// TIA Portal project "trafik_lamba_uygulama_sim" (V14)

(* hardware
DEVICE "S71500/ET200MP station_1"  S7-1500 station
   slot 0: "Rail_0"  Rack  6ES7 590-1***0-0AA0
   slot 1: "PLC_1"  CPU 1511C-1 PN  6ES7 511-1CK00-0AB0  V2.0
      slot 3: "CPU display_1"  6ES7591-1AA00-0AA0
*)

// ===== PLC "PLC_1"  CPU 1511C-1 PN =====

VAR_GLOBAL   // PLC tag table "Default tag table"
   ""start"" AT %I0.1 : Bool;
   ""reset"" AT %I0.0 : Bool;
   ""yol_1-3"" AT %Q0.0 : Bool;
   ""yol_2-4"" AT %Q0.1 : Bool;
   ""kirmizi_isik_yol-1"" AT %Q1.0 : Bool;
   ""sari_isik_yol-1"" AT %Q1.1 : Bool;
   ""yesil_isik_yol-1"" AT %Q1.2 : Bool;
   ""kirmizi_isik_yol-3"" AT %Q1.3 : Bool;
   ""sari_isik_yol-3"" AT %Q1.4 : Bool;
   ""yesil_isik_yol-3"" AT %Q1.5 : Bool;
   ""yol_5-6"" AT %Q0.2 : Bool;
   ""kirmizi_isik_yol-2"" AT %Q2.0 : Bool;
   ""sari_isik_yol-2"" AT %Q2.1 : Bool;
   ""yesil_isik_yol-2"" AT %Q2.2 : Bool;
   ""kirmizi_isik_yol-4"" AT %Q2.3 : Bool;
   ""sari_isik_yol-4"" AT %Q2.4 : Bool;
   ""yesil_isik_yol-4"" AT %Q2.5 : Bool;
   ""sistem"" AT %Q10.0 : Bool;
   ""yol_7-8"" AT %Q0.3 : Bool;
   ""kirmizi_isik_yol-5"" AT %Q3.0 : Bool;
   ""kirmizi_isik_yol-6"" AT %Q3.3 : Bool;
   ""sari_isik_yol-5"" AT %Q3.1 : Bool;
   ""sari_isik_yol-6"" AT %Q3.4 : Bool;
   ""yesil_isik_yol-5"" AT %Q3.2 : Bool;
   ""yesil_isik_yol-6"" AT %Q3.5 : Bool;
   ""kirmizi_isik_yol-7"" AT %Q4.0 : Bool;
   ""kirmizi_isik_yol-8"" AT %Q4.3 : Bool;
   ""sari_isik_yol-7"" AT %Q4.1 : Bool;
   ""sari_isik_yol-8"" AT %Q4.4 : Bool;
   ""yesil_isik_yol-7"" AT %Q4.2 : Bool;
   ""yesil_isik_yol-8"" AT %Q4.5 : Bool;
END_VAR